{attribute 'qualified_only'}
VAR_GLOBAL CONSTANT
	OPEN		: BOOL := FALSE;
	CLOSED		: BOOL := TRUE;
END_VAR

(* stored: Version 1.1.0.1
   GVL VALVE: Id {467d9cf7-3ac5-4d12-9df9-8ad9ce243200} *)
